// TIA Portal project "Tank Project Factory IO" (V15)
// Vorlageprojekt für das Buch mit Zielsystem S7-1200

(* hardware
DEVICE "S7-1200-Station_1"  S7-1200 Station
   slot 0: "Baugruppenträger_0"  Rack  V1.0
   slot 1: "PLC_1"  CPU 1211C DC/DC/DC  6ES7 211-1AE40-0XB0  V4.1
*)

// ===== PLC "PLC_1"  CPU 1211C DC/DC/DC =====

VAR_GLOBAL   // PLC tag table "Standard-Variablentabelle"
   "E Stop" AT %I0.0 : Bool;
   "Stop PB" AT %I0.1 : Bool;
   "Start PB" AT %I0.2 : Bool;
   "Reset PB" AT %I0.3 : Bool;
   "Fill PB" AT %I0.4 : Bool;
   "Drain PB" AT %I0.5 : Bool;
   "Auto" AT %I0.6 : Bool;
   "Manual" AT %I0.7 : Bool;
   "0% PB" AT %I1.0 : Bool;
   "25% PB" AT %I1.1 : Bool;
   "50% PB" AT %I1.2 : Bool;
   "75% PB" AT %I1.3 : Bool;
   "100% PB" AT %I1.4 : Bool;
   "Tank Level Sensor" AT %ID34 : Real;
   "0% Light" AT %Q0.0 : Bool;
   "25% Light" AT %Q0.1 : Bool;
   "50% Light" AT %Q0.2 : Bool;
   "75% Light" AT %Q0.3 : Bool;
   "100 % Light" AT %Q0.4 : Bool;
   "Reset Light" AT %Q0.5 : Bool;
   "Fill Light" AT %Q0.6 : Bool;
   "Drain Light" AT %Q0.7 : Bool;
   "Start Light" AT %Q1.0 : Bool;
   "Stop Light" AT %Q1.1 : Bool;
   "Fill Valve" AT %QD30 : Real;
   "Drain Valve" AT %QD34 : Real;
   "Sys Run" AT %M0.0 : Bool;
   "Emergency Stop" AT %M0.1 : Bool;
   "Clock_Byte" AT %MB10 : Byte;
   "Clock_10Hz" AT %M10.0 : Bool;
   "Clock_5Hz" AT %M10.1 : Bool;
   "Clock_2.5Hz" AT %M10.2 : Bool;
   "Clock_2Hz" AT %M10.3 : Bool;
   "Clock_1.25Hz" AT %M10.4 : Bool;
   "Clock_1Hz" AT %M10.5 : Bool;
   "Clock_0.625Hz" AT %M10.6 : Bool;
   "Clock_0.5Hz" AT %M10.7 : Bool;
   "Manual Mode" AT %M0.2 : Bool;
   "Auto Mode" AT %M0.3 : Bool;
   "Reset Mode" AT %M0.4 : Bool;
   "Auto Fill" AT %M0.5 : Bool;
   "Auto Drain" AT %M0.6 : Bool;
   "Fill level" AT %MD30 : DWord;
END_VAR

// folder: System blocks/Program resources

DATA_BLOCK "Reset Timer"   // DB1
{ S7_Optimized_Access := 'TRUE' }
AUTHOR : Simatic
FAMILY : IEC
NAME : IEC_TMR
VERSION : 1.0
// stored: InstanceOfName IEC_TIMER
"IEC_TIMER"
BEGIN
END_DATA_BLOCK

// folder: (top level)

FUNCTION "MHJ-PLC-Lab-Function-S71200" : Void   // FC9000, SCL
{ S7_Optimized_Access := 'TRUE' }
VERSION : 0.1
   VAR_TEMP
      rdTimeReturn : Int;
      outputTime : DTL;
      SyncVal : Byte;
      forVal : Int;
      forVal_2 : Int;
      Value : Byte;
   END_VAR
   VAR CONSTANT
      CompVal : Byte := 16#34;
      Value_01 : Byte := 16#11;
      Value_01_DW : DWord := 16#A165_D992;
      Value_02_DW : DWord := 16#58BE_4401;
   END_VAR
BEGIN

   #Value:=PEEK(area := 16#82,
        dbNumber := 0,
        byteOffset := 511);
   #Value := #Value + 1;

   POKE(area := 16#82,
        dbNumber := 0,
        byteOffset := 511,
        value := #Value);

   POKE(area:=16#81,
        dbNumber:=0,
        byteOffset:=1016,
        value:=#Value_01_DW);
   POKE(area := 16#81,
        dbNumber := 0,
        byteOffset := 1020,
        value := #Value_02_DW);

   POKE(area := 16#81,
        dbNumber := 0,
        byteOffset := 511,
        value := B#16#00);

   FOR #forVal := 0 TO 120 DO
       FOR #forVal_2:=0 TO 10 DO
           #rdTimeReturn:=RD_SYS_T(#outputTime);
           #rdTimeReturn := WR_SYS_T(#outputTime);
           #rdTimeReturn := RD_SYS_T(#outputTime);
           #rdTimeReturn := WR_SYS_T(#outputTime);
       END_FOR;
       #SyncVal:= PEEK(area := 16#81,
                      dbNumber := 0,
                      byteOffset := 511);
       IF #SyncVal = #CompVal THEN
          GOTO M_1;
       END_IF;
   END_FOR;
   RETURN;

   M_1:
   POKE(area := 16#81,
        dbNumber := 0,
        byteOffset := 511,
        value := B#16#0);
END_FUNCTION

ORGANIZATION_BLOCK "Main"   // OB1, FBD, ProgramCycle
TITLE = "Main Program Sweep (Cycle)"
{ S7_Optimized_Access := 'TRUE' }
VERSION : 0.1
   VAR_INPUT
      Initial_Call : Bool;   // Initial call of this OB
      Remanence : Bool;   // =True, if remanent data are available
   END_VAR
BEGIN

REGION Network 1: Konnektierungsbaustein für PLC-Lab
   // Im Netzwerk 1 wird der Konnektierungsbaustein für PLC-Lab aufgerufen.
   // Dieser Aufruf darf nicht entfernt werden!
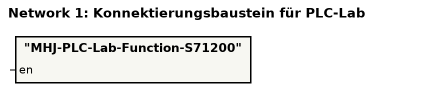
   "MHJ-PLC-Lab-Function-S71200"();
END_REGION

REGION Network 2: Ihr Programm
   // Schreiben Sie ab Netzwerk 2 Ihr Programm
END_REGION
END_ORGANIZATION_BLOCK

ORGANIZATION_BLOCK "Main_1"   // OB123, LAD, ProgramCycle
TITLE = "Main Program Sweep (Cycle)"
{ S7_Optimized_Access := 'TRUE' }
VERSION : 0.1
   VAR_INPUT
      Initial_Call : Bool;   // Initial call of this OB
      Remanence : Bool;   // =True, if remanent data are available
   END_VAR
   VAR_TEMP   // added for the SCL form of the ladder/FBD networks
      _w1 : Bool;
   END_VAR
BEGIN

REGION Network 1
   // System Run Instruction
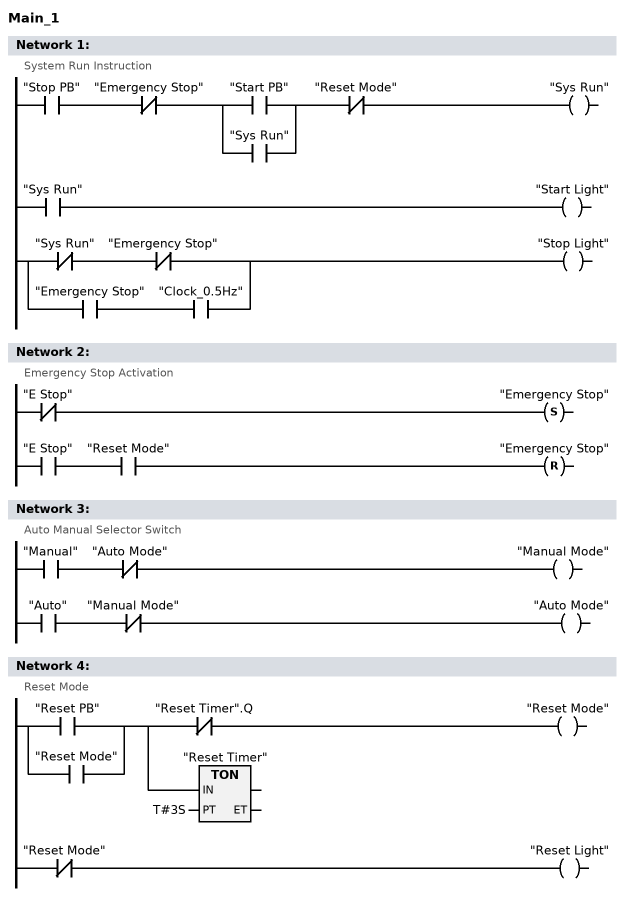
   RUNG wire#powerrail
      Contact( "Stop PB" )
      I_Contact( "Emergency Stop" )
      wire#w1
      Contact( "Start PB" )
      wire#w2
      I_Contact( "Reset Mode" )
      Coil( "Sys Run" )
   END_RUNG
   RUNG wire#w1
      Contact( "Sys Run" )
   END_RUNG wire#w2
   RUNG wire#powerrail
      Contact( "Sys Run" )
      Coil( "Start Light" )
   END_RUNG
   RUNG wire#powerrail
      I_Contact( "Sys Run" )
      I_Contact( "Emergency Stop" )
      wire#w3
      Coil( "Stop Light" )
   END_RUNG
   RUNG wire#powerrail
      Contact( "Emergency Stop" )
      Contact( "Clock_0.5Hz" )
   END_RUNG wire#w3
   // the same network as SCL:
   "Sys Run" := "Stop PB" AND NOT "Emergency Stop" AND ("Start PB" OR "Sys Run") AND NOT "Reset Mode";
   "Start Light" := "Sys Run";
   "Stop Light" := (NOT "Sys Run" AND NOT "Emergency Stop") OR ("Emergency Stop" AND "Clock_0.5Hz");
END_REGION

REGION Network 2
   // Emergency Stop Activation
   RUNG wire#powerrail
      I_Contact( "E Stop" )
      S_Coil( "Emergency Stop" )
   END_RUNG
   RUNG wire#powerrail
      Contact( "E Stop" )
      Contact( "Reset Mode" )
      R_Coil( "Emergency Stop" )
   END_RUNG
   // the same network as SCL:
   IF NOT "E Stop" THEN "Emergency Stop" := TRUE; END_IF;
   IF "E Stop" AND "Reset Mode" THEN "Emergency Stop" := FALSE; END_IF;
END_REGION

REGION Network 3
   // Auto Manual Selector Switch
   RUNG wire#powerrail
      Contact( "Manual" )
      I_Contact( "Auto Mode" )
      Coil( "Manual Mode" )
   END_RUNG
   RUNG wire#powerrail
      Contact( "Auto" )
      I_Contact( "Manual Mode" )
      Coil( "Auto Mode" )
   END_RUNG
   // the same network as SCL:
   "Manual Mode" := "Manual" AND NOT "Auto Mode";
   "Auto Mode" := "Auto" AND NOT "Manual Mode";
END_REGION

REGION Network 4
   // Reset Mode
   #_w1 := "Reset PB" OR "Reset Mode";
   "Reset Mode" := #_w1 AND NOT "Reset Timer".Q;
   "Reset Timer".TON(IN := #_w1, PT := T#3S);
   "Reset Light" := NOT "Reset Mode";
END_REGION
END_ORGANIZATION_BLOCK

ORGANIZATION_BLOCK "Manual Fill & Drain"   // OB124, LAD, ProgramCycle
TITLE = "Main Program Sweep (Cycle)"
{ S7_Optimized_Access := 'TRUE' }
VERSION : 0.1
   VAR_INPUT
      Initial_Call : Bool;   // Initial call of this OB
      Remanence : Bool;   // =True, if remanent data are available
   END_VAR
   VAR_TEMP   // added for the SCL form of the ladder/FBD networks
      _w1 : Bool;
   END_VAR
BEGIN

REGION Network 1
   // Manual Fill
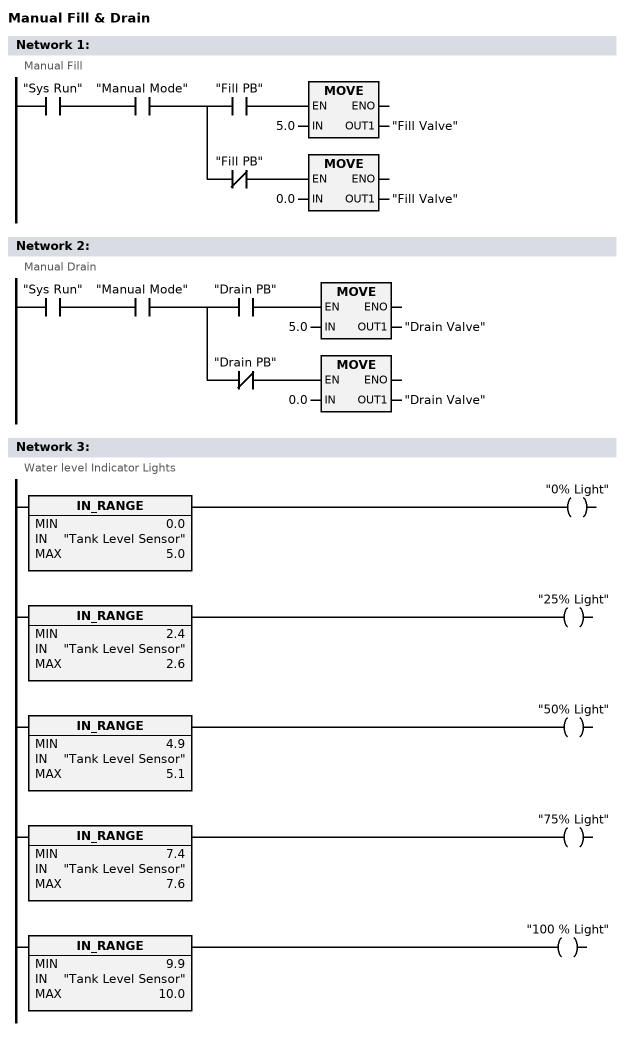
   RUNG wire#powerrail
      Contact( "Sys Run" )
      Contact( "Manual Mode" )
      wire#w1
      Contact( "Fill PB" )
      Move(in := 5.0, out1 => "Fill Valve")
   END_RUNG
   RUNG wire#w1
      I_Contact( "Fill PB" )
      Move(in := 0.0, out1 => "Fill Valve")
   END_RUNG
   // the same network as SCL:
   #_w1 := "Sys Run" AND "Manual Mode";
   IF #_w1 AND "Fill PB" THEN "Fill Valve" := 5.0; END_IF;
   IF #_w1 AND NOT "Fill PB" THEN "Fill Valve" := 0.0; END_IF;
END_REGION

REGION Network 2
   // Manual Drain
   RUNG wire#powerrail
      Contact( "Sys Run" )
      Contact( "Manual Mode" )
      wire#w1
      Contact( "Drain PB" )
      Move(in := 5.0, out1 => "Drain Valve")
   END_RUNG
   RUNG wire#w1
      I_Contact( "Drain PB" )
      Move(in := 0.0, out1 => "Drain Valve")
   END_RUNG
   // the same network as SCL:
   #_w1 := "Sys Run" AND "Manual Mode";
   IF #_w1 AND "Drain PB" THEN "Drain Valve" := 5.0; END_IF;
   IF #_w1 AND NOT "Drain PB" THEN "Drain Valve" := 0.0; END_IF;
END_REGION

REGION Network 3
   // Water level Indicator Lights
   RUNG wire#powerrail
      { S7_Templates := "SrcType := Real" } InRange(min := 0.0, in := "Tank Level Sensor", max := 5.0)
      Coil( "0% Light" )
   END_RUNG
   RUNG wire#powerrail
      { S7_Templates := "SrcType := Real" } InRange(min := 2.4, in := "Tank Level Sensor", max := 2.6)
      Coil( "25% Light" )
   END_RUNG
   RUNG wire#powerrail
      { S7_Templates := "SrcType := Real" } InRange(min := 4.9, in := "Tank Level Sensor", max := 5.1)
      Coil( "50% Light" )
   END_RUNG
   RUNG wire#powerrail
      { S7_Templates := "SrcType := Real" } InRange(min := 7.4, in := "Tank Level Sensor", max := 7.6)
      Coil( "75% Light" )
   END_RUNG
   RUNG wire#powerrail
      { S7_Templates := "SrcType := Real" } InRange(min := 9.9, in := "Tank Level Sensor", max := 10.0)
      Coil( "100 % Light" )
   END_RUNG
   // the same network as SCL:
   "0% Light" := (0.0 <= "Tank Level Sensor") AND ("Tank Level Sensor" <= 5.0);
   "25% Light" := (2.4 <= "Tank Level Sensor") AND ("Tank Level Sensor" <= 2.6);
   "50% Light" := (4.9 <= "Tank Level Sensor") AND ("Tank Level Sensor" <= 5.1);
   "75% Light" := (7.4 <= "Tank Level Sensor") AND ("Tank Level Sensor" <= 7.6);
   "100 % Light" := (9.9 <= "Tank Level Sensor") AND ("Tank Level Sensor" <= 10.0);
END_REGION
END_ORGANIZATION_BLOCK

ORGANIZATION_BLOCK "Auto Fill & Drain"   // OB125, LAD, ProgramCycle
TITLE = "Main Program Sweep (Cycle)"
{ S7_Optimized_Access := 'TRUE' }
VERSION : 0.1
   VAR_INPUT
      Initial_Call : Bool;   // Initial call of this OB
      Remanence : Bool;   // =True, if remanent data are available
   END_VAR
BEGIN

REGION Network 1
   // Auto Fill and Drain
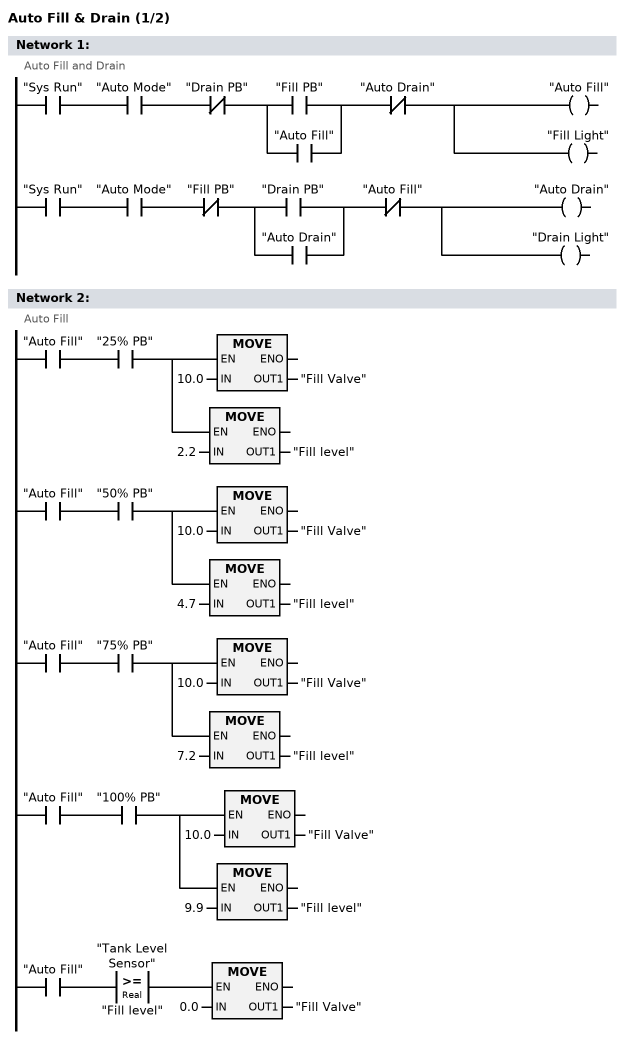
   RUNG wire#powerrail
      Contact( "Sys Run" )
      Contact( "Auto Mode" )
      I_Contact( "Drain PB" )
      wire#w1
      Contact( "Fill PB" )
      wire#w2
      I_Contact( "Auto Drain" )
      wire#w3
      Coil( "Auto Fill" )
   END_RUNG
   RUNG wire#w1
      Contact( "Auto Fill" )
   END_RUNG wire#w2
   RUNG wire#w3
      Coil( "Fill Light" )
   END_RUNG
   RUNG wire#powerrail
      Contact( "Sys Run" )
      Contact( "Auto Mode" )
      I_Contact( "Fill PB" )
      wire#w4
      Contact( "Drain PB" )
      wire#w5
      I_Contact( "Auto Fill" )
      wire#w6
      Coil( "Auto Drain" )
   END_RUNG
   RUNG wire#w4
      Contact( "Auto Drain" )
   END_RUNG wire#w5
   RUNG wire#w6
      Coil( "Drain Light" )
   END_RUNG
   // the same network as SCL:
   "Auto Fill" := "Sys Run" AND "Auto Mode" AND NOT "Drain PB" AND ("Fill PB" OR "Auto Fill") AND NOT "Auto Drain";
   "Fill Light" := "Auto Fill";
   "Auto Drain" := "Sys Run" AND "Auto Mode" AND NOT "Fill PB" AND ("Drain PB" OR "Auto Drain") AND NOT "Auto Fill";
   "Drain Light" := "Auto Drain";
END_REGION

REGION Network 2
   // Auto Fill
   RUNG wire#powerrail
      Contact( "Auto Fill" )
      Contact( "25% PB" )
      wire#w1
      Move(in := 10.0, out1 => "Fill Valve")
   END_RUNG
   RUNG wire#w1
      Move(in := 2.2, out1 => "Fill level")
   END_RUNG
   RUNG wire#powerrail
      Contact( "Auto Fill" )
      Contact( "50% PB" )
      wire#w2
      Move(in := 10.0, out1 => "Fill Valve")
   END_RUNG
   RUNG wire#w2
      Move(in := 4.7, out1 => "Fill level")
   END_RUNG
   RUNG wire#powerrail
      Contact( "Auto Fill" )
      Contact( "75% PB" )
      wire#w3
      Move(in := 10.0, out1 => "Fill Valve")
   END_RUNG
   RUNG wire#w3
      Move(in := 7.2, out1 => "Fill level")
   END_RUNG
   RUNG wire#powerrail
      Contact( "Auto Fill" )
      Contact( "100% PB" )
      wire#w4
      Move(in := 10.0, out1 => "Fill Valve")
   END_RUNG
   RUNG wire#w4
      Move(in := 9.9, out1 => "Fill level")
   END_RUNG
   RUNG wire#powerrail
      Contact( "Auto Fill" )
      { S7_Templates := "SrcType := Real" } GE_Contact(in1 := "Tank Level Sensor", in2 := "Fill level")
      Move(in := 0.0, out1 => "Fill Valve")
   END_RUNG
   // the same network as SCL:
   IF "Auto Fill" AND "25% PB" THEN
       "Fill Valve" := 10.0;
       "Fill level" := 2.2;
   END_IF;
   IF "Auto Fill" AND "50% PB" THEN
       "Fill Valve" := 10.0;
       "Fill level" := 4.7;
   END_IF;
   IF "Auto Fill" AND "75% PB" THEN
       "Fill Valve" := 10.0;
       "Fill level" := 7.2;
   END_IF;
   IF "Auto Fill" AND "100% PB" THEN
       "Fill Valve" := 10.0;
       "Fill level" := 9.9;
   END_IF;
   IF "Auto Fill" AND ("Tank Level Sensor" >= "Fill level") THEN "Fill Valve" := 0.0; END_IF;
END_REGION

REGION Network 3
   // Auto Drain
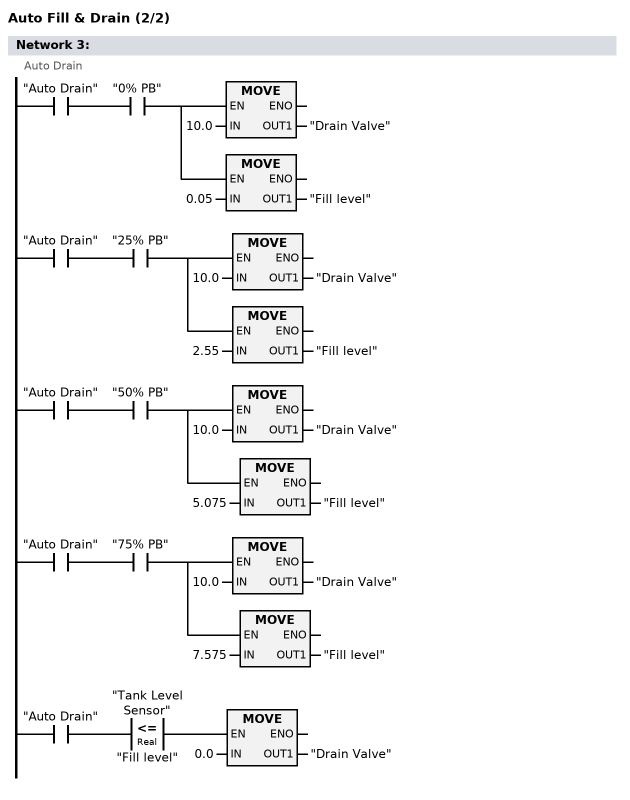
   RUNG wire#powerrail
      Contact( "Auto Drain" )
      Contact( "0% PB" )
      wire#w1
      Move(in := 10.0, out1 => "Drain Valve")
   END_RUNG
   RUNG wire#w1
      Move(in := 0.05, out1 => "Fill level")
   END_RUNG
   RUNG wire#powerrail
      Contact( "Auto Drain" )
      Contact( "25% PB" )
      wire#w2
      Move(in := 10.0, out1 => "Drain Valve")
   END_RUNG
   RUNG wire#w2
      Move(in := 2.55, out1 => "Fill level")
   END_RUNG
   RUNG wire#powerrail
      Contact( "Auto Drain" )
      Contact( "50% PB" )
      wire#w3
      Move(in := 10.0, out1 => "Drain Valve")
   END_RUNG
   RUNG wire#w3
      Move(in := 5.075, out1 => "Fill level")
   END_RUNG
   RUNG wire#powerrail
      Contact( "Auto Drain" )
      Contact( "75% PB" )
      wire#w4
      Move(in := 10.0, out1 => "Drain Valve")
   END_RUNG
   RUNG wire#w4
      Move(in := 7.575, out1 => "Fill level")
   END_RUNG
   RUNG wire#powerrail
      Contact( "Auto Drain" )
      { S7_Templates := "SrcType := Real" } LE_Contact(in1 := "Tank Level Sensor", in2 := "Fill level")
      Move(in := 0.0, out1 => "Drain Valve")
   END_RUNG
   // the same network as SCL:
   IF "Auto Drain" AND "0% PB" THEN
       "Drain Valve" := 10.0;
       "Fill level" := 0.05;
   END_IF;
   IF "Auto Drain" AND "25% PB" THEN
       "Drain Valve" := 10.0;
       "Fill level" := 2.55;
   END_IF;
   IF "Auto Drain" AND "50% PB" THEN
       "Drain Valve" := 10.0;
       "Fill level" := 5.075;
   END_IF;
   IF "Auto Drain" AND "75% PB" THEN
       "Drain Valve" := 10.0;
       "Fill level" := 7.575;
   END_IF;
   IF "Auto Drain" AND ("Tank Level Sensor" <= "Fill level") THEN "Drain Valve" := 0.0; END_IF;
END_REGION
END_ORGANIZATION_BLOCK